TYPE ST_IO2_SingleInputCtrl :
STRUCT
	eTypeInput 		: E_IO2_Type;
	tTimeOnFilter		: TIME;
	tTimeOffFilter 		: TIME;
	sInputName		: STRING(40);
END_STRUCT
END_TYPE

(* stored: Version 1.1.0.1
   DUT ST_IO2_SingleInputCtrl: Id {5287dd9b-b574-4b74-96d1-243a0abf172b} *)
